FUNCTION POU_MoveToPos : INT
VAR_INPUT
	actualPos : INT ;
	requiredPos : INT;
	speed: INT;

	
END_VAR
VAR
	timer : ton;
	newPos : int;
	startTimer: BOOL;
	calculatedTime: time;
END_VAR

calculatedTime :=INT_TO_TIME(1000/speed);
timer(in:= startTimer, pt:= calculatedTime);
startTimer:= TRUE;
IF timer.Q THEN
	startTimer:=FALSE;
	IF requiredPos < actualpos THEN
		newpos := actualPos -1;
	ELSIF requiredpos > actualpos THEN
		newpos := actualPos +1; 
	END_IF
END_IF

END_FUNCTION

(* stored: Version 1.1.0.1, ProductVersion 3.1.4024.12
   POU POU_MoveToPos: Id {f1b905d7-21a7-4edb-bcb9-64fac2a8debd}, SpecialFunc None *)
